FUNCTION_BLOCK TcAbbLinkin
VAR_INPUT
	_connectionEnabled : BOOL := TRUE;
END_VAR
VAR_OUTPUT
END_VAR
VAR
	_httpClient: FB_IotHttpClient;
END_VAR

METHOD ConnectionStart : BOOL
VAR_INPUT
	connectionConfig:	AbbLinkinConnectionConfig_Typ;	
END_VAR


// Configuration
_httpClient.sHostName := connectionConfig.remoteIpAddress;
_httpClient.nHostPort := connectionConfig.remotePort;
_httpClient.bKeepAlive := TRUE;
_httpClient.tConnectionTimeout := T#10S;


CASE connectionConfig.rwsVersion OF
	ABBLINKIN_RWS_API_VERSION.V1:
		_httpClient.stTLS.bNoServerCertCheck := TRUE;
		
	ABBLINKIN_RWS_API_VERSION.V2:
		_httpClient.stTLS.bNoServerCertCheck := FALSE;
		// TODO: add other tls settings
END_CASE



_connectionEnabled := TRUE;
END_METHOD

METHOD ConnectionStop : BOOL
VAR_INPUT
END_VAR

_connectionEnabled := FALSE;
END_METHOD

METHOD GetIO : BOOL
VAR_INPUT
END_VAR
END_METHOD

METHOD GetState : BOOL
VAR_INPUT
END_VAR
END_METHOD

METHOD GetSymbol : BOOL
VAR_INPUT
END_VAR
END_METHOD

METHOD IOWatchInit : BOOL
VAR_INPUT
END_VAR
END_METHOD

METHOD MotorsOff : BOOL
VAR_INPUT
END_VAR
END_METHOD

METHOD MotorsOn : BOOL
VAR_INPUT
END_VAR
END_METHOD

METHOD PowerOff : BOOL
VAR_INPUT
END_VAR
END_METHOD

METHOD PowerOn : BOOL
VAR_INPUT
END_VAR
END_METHOD

METHOD RapidReset : BOOL
VAR_INPUT
END_VAR
END_METHOD

METHOD RapidStart : BOOL
VAR_INPUT
END_VAR
END_METHOD

METHOD RapidStop : BOOL
VAR_INPUT
END_VAR
END_METHOD

METHOD SetIO : BOOL
VAR_INPUT
END_VAR
END_METHOD

METHOD SetSymbol : BOOL
VAR_INPUT
END_VAR
END_METHOD

END_FUNCTION_BLOCK

(* stored: Version 1.1.0.1, ProductVersion 3.1.4024.12
   POU TcAbbLinkin: Id {83aacf3c-7637-43d5-b1b4-45d5caf263aa}, SpecialFunc None
   Method ConnectionStart: Id {ae04014b-99d1-4864-b820-dd29eedcb99e}
   Method ConnectionStop: Id {fb28cdfe-8e1b-44f1-869a-b019fa3c0b7f}
   Method GetIO: Id {bd29dab4-cb08-45fe-84ff-e3737f6110e8}
   Method GetState: Id {39878dda-bc14-4b8b-833d-1d9c4ab2cc84}
   Method GetSymbol: Id {85af9ad1-0b82-4752-9ea8-7aabc8bae9aa}
   Method IOWatchInit: Id {73cfccc7-56e4-4d35-a07c-3dccb64e2e07}
   Method MotorsOff: Id {0e9c796b-4548-4647-8b3c-207480990c05}
   Method MotorsOn: Id {61a3e16c-d842-4ebd-be26-10100c74cc52}
   Method PowerOff: Id {7e704635-bfa1-4267-9db0-7f188918765f}
   Method PowerOn: Id {e270cd96-8004-4691-9cb0-f9c8d0300c0b}
   Method RapidReset: Id {8680bb07-92fa-45e4-93ac-a5f26d92aefb}
   Method RapidStart: Id {2acbd226-93a7-4d9b-8ddf-34c3d2ee1221}
   Method RapidStop: Id {648edf84-4daf-4e8c-8ad5-61b6305b08fb}
   Method SetIO: Id {ce5e4a58-9783-46a9-ba0d-44594affd7f4}
   Method SetSymbol: Id {bc0a5da5-b662-4b6f-a5f4-f2caf9d05bbf} *)
